PROGRAM P_Demo_F_BA_IsWeekdayValid
VAR
    argEDay                        : E_BA_Weekday                  ; // eDay
    fnReturn                       : BOOL; // 返回值
END_VAR

// =============================================================================
// Tc3_BA2_Common.F_BA_IsWeekdayValid 演示程序
// =============================================================================
// 场景：配置导入校验。
//
// 价值：同其它 IsValid 系列。
//
// 验证：登录 PLC 后，按例程内变量在线写值；监视输出 / 返回值，结合 §1 功能
//       简述的预期行为对照（详见配套 .md 文档 §7 业务场景）。
//
// 验证步骤：
//   1. 右键 PLC 项目下 POUs 文件夹 → Add → Existing Item → 选本 .TcPOU 文件
//   2. 引用 Tc3_BA2_Common（References → Add library）
//   3. 编译 → 登录 → 运行；按上方『验证』指引在线写值观察
// =============================================================================

fnReturn := F_BA_IsWeekdayValid(
    eDay                     := argEDay
);

END_PROGRAM

(* stored: Version 1.1.0.1, ProductVersion 3.1.4024.5
   POU P_Demo_F_BA_IsWeekdayValid: Id {78bfb6d5-5925-5f03-b12e-734582ff19ff}, SpecialFunc None *)
